TYPE StepLog :
STRUCT
	config 		: StepConfig;
	status		: StepStatus;
END_STRUCT
END_TYPE

(* stored: Version 1.1.0.1, ProductVersion 3.1.4024.11
   DUT StepLog: Id {f5ed18f1-5a72-4876-aafe-12a27ea0d0b4} *)
